// Output from safety check task
// Input to master arm control task
TYPE ST_SafetyData :
STRUCT
	m_slaveErrFlag :ARRAY[1..g_sArmNum] OF BOOL :=[4(FALSE)];
	m_setupErrFlag :ARRAY[1..g_sArmNum] OF BOOL :=[4(FALSE)];
	m_cartErrFlag :BOOL :=FALSE;
	m_cartSteadyFootErr :BOOL;
	m_cartWheelErr :BOOL;
	m_cartStandColumnErr :BOOL;
	m_cartAdjustErr :BOOL;
	m_cartOverhangErr :BOOL;
END_STRUCT
END_TYPE

(* stored: Version 1.1.0.1, ProductVersion 3.1.4024.11
   DUT ST_SafetyData: Id {322b279b-f9a5-4da8-8f90-8d4b82ec3137} *)
